// TIA Portal V18 export
TYPE "PLCtoMES_MainCheckIn_ext"
// stored: IsFailsafeCompliant false
   STRUCT
      Load_Station1ChickInReq : Bool;   // 本站工位1主零件过站查询事件触发位
      Load_Station2ChickInReq : Bool;   // 本站工位2主零件过站查询事件触发位
      Load_Station3ChickInReq : Bool;   // 本站工位3主零件过站查询事件触发位
      Load_Station4ChickInReq : Bool;   // 本站工位4主零件过站查询事件触发位
      Load_Station5ChickInReq : Bool;   // 本站工位5主零件过站查询事件触发位
      Load_Station6ChickInReq : Bool;   // 本站工位6主零件过站查询事件触发位
      Load_Station7ChickInReq : Bool;   // 本站工位7主零件过站查询事件触发位
      Load_Station8ChickInReq : Bool;   // 本站工位8主零件过站查询事件触发位
   END_STRUCT;
END_TYPE
